{attribute 'qualified_only'}
TYPE ErrorCodeEnum :
(
	undefined := 0,
  invalidInput,
  synchronizationCalculation,
  calculateStep1Failed
);
END_TYPE

(* stored: Version 1.1.0.1, ProductVersion 3.1.4024.9
   DUT ErrorCodeEnum: Id {b6f9027e-b647-46b0-a8f4-fdacb3d850bf} *)
